Staubli VAL3: espanol.dtx

public string Yes = "Yes "
public string No = "No"
